(* IEC 61131-3 sources: SRCI/RobotLibrary/RobotLibrary/POUs/SearchHardstop/MC_SearchHardStop, 1 file *)

(* ---- MC_SearchHardStopFB.st ---- *)
/// Move robot into contact with obstruction (mechanical Limit) and hold it in this position
FUNCTION_BLOCK MC_SearchHardStopFB EXTENDS RobotLibraryBaseExecuteFB
// -------------------------------------------------------------------------
//  SRCI Robot Library
// -------------------------------------------------------------------------
//
//  Object:      SearchHardStopFB
//  Author:      Thorsten Brach
//  Date:        2024-06-01
//
//  Description:
//
//
//  Copyright:
//    (C) 2024 Thorsten Brach. All rights reserved
//             Licensed under the LGPL-3.0 license.
//
//  Disclaimer:
//    This project is provided without any guarantee and can be used for
//    private and commercial purposes. Any use is at the user’s
//    own risk and responsibility.
//
// -------------------------------------------------------------------------
VAR_INPUT
  /// Parameter which determines the behavior towards the previously sent and still active or buffered commands
  AbortingMode       : AbortingMode;
  /// Defines the target sequence in which the command will be executed
  SequenceFlag       : SequenceFlag;
  /// command parameter
  ParCmd             : SearchHardStopParCmd;
END_VAR

VAR_OUTPUT
  /// Command is transferred and confirmed by the RC
  CommandBuffered    : BOOL;
  /// The command takes control of the motion of the according axis group
  Active             : BOOL;
  /// The command was aborted by another command.
  CommandAborted     : BOOL;
  /// TRUE, while command is interrupted during execution and can be continued
  CommandInterrupted : BOOL;
  /// command results
  OutCmd             : SearchHardStopOutCmd;
END_VAR

VAR
  /// internal copy of command parameter
 _parCmd             : SearchHardStopParCmd;
  /// command data to send
 _command            : SearchHardStopSendData;
  /// response data received
 _response           : SearchHardStopRecvData;
END_VAR

  SUPER^(AxesGroup := AxesGroup);

END_FUNCTION_BLOCK

METHOD CheckParameterChanged : BOOL
VAR_IN_OUT
  /// Robot assignment of function
  AxesGroup    : AxesGroup;
END_VAR

  // Check ParCmd Size is > 0, becaue MemCmp does not work correctly with size = 0
  IF (SIZEOF(ParCmd) = 0)
  THEN
    RETURN;
  END_IF

  // compare memory
  CheckParameterChanged := ( MemCmp(ADR(ParCmd), ADR(_parCmd), SIZEOF(ParCmd)) <> RobotLibraryConstants.OK );

  IF ( CheckParameterChanged )
  THEN
    // update internal copy of parameters
   _parCmd := ParCmd;
    // inc parameter sequence
   _command.ParSeq := _command.ParSeq + 1;
    // update command data
    CommandData := CreateCommandPayload(); // ( Access via reference to rCommandFB in ACR )
    // notify active command register
    AxesGroup.Acyclic.ActiveCommandRegister.NotifyParameterChanged := _uniqueID;
  END_IF

END_METHOD

METHOD INTERNAL CreateCommandPayload : SendData
// Table 6-405: Sent CMD payload (PLC to RC) of "SearchHardStop"
// --------------------------
// Header
// --------------------------
// Byte 00 : UINT  - Type HB
// Byte 01 :       - Type LB
// Byte 02 : USINT - Reserve | ExecutionMode
// Byte 03 : USINT - ParSeq  | Priority
// --------------------------
// Datablock
// --------------------------
 // Byte 04 : UINT  VelocityRate;
 // Byte 05 :       VelocityRate;
 // Byte 06 : UINT  AccelerationRate;
 // Byte 07 :       AccelerationRate;
 // Byte 08 : UINT  DecelerationRate;
 // Byte 09 :       DecelerationRate;
 // Byte 10 : UINT  JerkRate;
 // Byte 11 :       JerkRate;
 // Byte 12 : USINT ToolNo;
 // Byte 13 : USINT FrameNo;
 // Byte 14 : REAL  Position.X;
 // Byte 15 :       Position.X;
 // Byte 16 :       Position.X;
 // Byte 17 :       Position.X;
 // Byte 18 : REAL  Position.Y;
 // Byte 19 :       Position.Y;
 // Byte 20 :       Position.Y;
 // Byte 21 :       Position.Y;
 // Byte 22 : REAL  Position.Z;
 // Byte 23 :       Position.Z;
 // Byte 24 :       Position.Z;
 // Byte 25 :       Position.Z;
 // Byte 26 : REAL  Position.RX;
 // Byte 27 :       Position.RX;
 // Byte 28 :       Position.RX;
 // Byte 29 :       Position.RX;
 // Byte 30 : REAL  Position.RY;
 // Byte 31 :       Position.RY;
 // Byte 32 :       Position.RY;
 // Byte 33 :       Position.RY;
 // Byte 34 : REAL  Position.RZ;
 // Byte 35 :       Position.RZ;
 // Byte 36 :       Position.RZ;
 // Byte 37 :       Position.RZ;
 // Byte 38 : BYTE  - - - - - W E S;
 // Byte 39 : BYTE  Reserved;
 // Byte 40 : BYTE  Position.TurnNumber[0];
 // Byte 41 : BYTE  Position.TurnNumber[1];
 // Byte 42 : BYTE  Position.TurnNumber[2];
 // Byte 43 : BYTE  Position.TurnNumber[3];
 // Byte 44 : REAL  Position.E1;
 // Byte 45 :       Position.E1;
 // Byte 46 :       Position.E1;
 // Byte 47 :       Position.E1;
 // Byte 48 : USINT OriMode;
 // Byte 49 : USINT DetectionMode;
 // Byte 50 : BOOL  Manipulation;
 // Byte 51 : BYTE  Reserved;
 // Byte 52 : REAL  DetectionVector[0];
 // Byte 53 :       DetectionVector[0];
 // Byte 54 :       DetectionVector[0];
 // Byte 55 :       DetectionVector[0];
 // Byte 56 : REAL  DetectionVector[1];
 // Byte 57 :       DetectionVector[1];
 // Byte 58 :       DetectionVector[1];
 // Byte 59 :       DetectionVector[1];
 // Byte 60 : REAL  DetectionVector[2];
 // Byte 61 :       DetectionVector[2];
 // Byte 62 :       DetectionVector[2];
 // Byte 63 :       DetectionVector[2];
 // Byte 64 : REAL  DetectionVector[3];
 // Byte 65 :       DetectionVector[3];
 // Byte 66 :       DetectionVector[3];
 // Byte 67 :       DetectionVector[3];
 // Byte 68 : REAL  DetectionVector[4];
 // Byte 69 :       DetectionVector[4];
 // Byte 70 :       DetectionVector[4];
 // Byte 71 :       DetectionVector[4];
 // Byte 72 : REAL  DetectionVector[5];
 // Byte 73 :       DetectionVector[5];
 // Byte 74 :       DetectionVector[5];
 // Byte 75 :       DetectionVector[5];
 // Byte 76 : BYTE  ConfigMode[0];
 // Byte 77 : BYTE  ConfigMode[1];
 // Byte 78 : USINT TurnMode;
 // Byte 79 : REAL  Position.E2;
 // Byte 80 :       Position.E2;
 // Byte 81 :       Position.E2;
 // Byte 82 :       Position.E2;
 // Byte 83 : REAL  Position.E3;
 // Byte 84 :       Position.E3;
 // Byte 85 :       Position.E3;
 // Byte 86 :       Position.E3;
 // Byte 87 : REAL  Position.E4;
 // Byte 88 :       Position.E4;
 // Byte 89 :       Position.E4;
 // Byte 90 :       Position.E4;
 // Byte 91 : REAL  Position.E5;
 // Byte 92 :       Position.E5;
 // Byte 93 :       Position.E5;
 // Byte 94 :       Position.E5;
 // Byte 95 : REAL  Position.E6;
 // Byte 96 :       Position.E6;
 // Byte 97 :       Position.E6;
 // Byte 98 :       Position.E6;

  // set command parameter
  _command.CmdTyp           :=  CmdType.SearchHardstop;
  _command.ExecMode         :=  ExecMode;
  _command.ParSeq           := _command.ParSeq;
  _command.Priority         :=  Priority;
  _command.VelocityRate     := REAL_TO_UINT(_parCmd.VelocityRate     * RobotLibraryConstants.REAL_CONVERSION_FACTOR);
  _command.AccelerationRate := REAL_TO_UINT(_parCmd.AccelerationRate * RobotLibraryConstants.REAL_CONVERSION_FACTOR);
  _command.DecelerationRate := REAL_TO_UINT(_parCmd.DecelerationRate * RobotLibraryConstants.REAL_CONVERSION_FACTOR);
  _command.JerkRate         := REAL_TO_UINT(_parCmd.JerkRate         * RobotLibraryConstants.REAL_CONVERSION_FACTOR);
  _command.ToolNo           := _parCmd.ToolNo;
  _command.FrameNo          := _parCmd.FrameNo;
  _command.Position         := _parCmd.Position;
  _command.OriMode          := _parCmd.OriMode;
  _command.DetectionMode    := _parCmd.DetectionMode;
  _command.Manipulation     := _parCmd.Manipulation;
  _command.Reserve          :=  0;
  _command.DetectionVector  := _parCmd.DetectionVector;
  _command.ConfigMode[0].0   := _parCmd.ConfigMode.Shoulder.0;
  _command.ConfigMode[0].1   := _parCmd.ConfigMode.Shoulder.1;
  _command.ConfigMode[0].2   := _parCmd.ConfigMode.Shoulder.2;
  _command.ConfigMode[0].3   := _parCmd.ConfigMode.Shoulder.3;
  _command.ConfigMode[0].4   := _parCmd.ConfigMode.Elbow.0;
  _command.ConfigMode[0].5   := _parCmd.ConfigMode.Elbow.1;
  _command.ConfigMode[0].6   := _parCmd.ConfigMode.Elbow.2;
  _command.ConfigMode[0].7   := _parCmd.ConfigMode.Elbow.3;
  _command.ConfigMode[1].0   := _parCmd.ConfigMode.Wrist.0;
  _command.ConfigMode[1].1   := _parCmd.ConfigMode.Wrist.1;
  _command.ConfigMode[1].2   := _parCmd.ConfigMode.Wrist.2;
  _command.ConfigMode[1].3   := _parCmd.ConfigMode.Wrist.3;
  _command.ConfigMode[1].4   := FALSE;
  _command.ConfigMode[1].5   := FALSE;
  _command.ConfigMode[1].6   := FALSE;
  _command.ConfigMode[1].7   := FALSE;
  _command.TurnMode         := _parCmd.TurnMode;

  // copy command data to header
  _cmdHeader := _command;
  // call base implementation to copy header to payload buffer
  CreateCommandPayload := SUPER^.CreateCommandPayload();

  // add command.VelocityRate
  CreateCommandPayload.AddUint(_command.VelocityRate);
  // add command.AccelerationRate
  CreateCommandPayload.AddUint(_command.AccelerationRate);
  // add command.DecelerationRate
  CreateCommandPayload.AddUint(_command.DecelerationRate);
  // add command.JerkRate
  CreateCommandPayload.AddUint(_command.JerkRate);
  // add command.ToolNo
  CreateCommandPayload.AddUsint(_command.ToolNo);
  // add command.FrameNo
  CreateCommandPayload.AddUsint(_command.FrameNo);
  // add command.Position.X
  CreateCommandPayload.AddReal(_command.Position.X);
  // add command.Position.Y
  CreateCommandPayload.AddReal(_command.Position.Y);
  // add command.Position.Z
  CreateCommandPayload.AddReal(_command.Position.Z);
  // add command.Position.Rx
  CreateCommandPayload.AddReal(_command.Position.Rx);
  // add command.Position.Ry
  CreateCommandPayload.AddReal(_command.Position.Ry);
  // add command.Position.Rz
  CreateCommandPayload.AddReal(_command.Position.Rz);
  // add command.Position.Config
  CreateCommandPayload.AddArmConfig(_command.Position.Config);
  // add command.Position.TurnNumber
  CreateCommandPayload.AddTurnNumber(_command.Position.TurnNumber);
  // add command.Position.E1
  CreateCommandPayload.AddReal(_command.Position.E1);
  // add command.OriMode
  CreateCommandPayload.AddUsint(_command.OriMode);
  // add command.DetectionMode
  CreateCommandPayload.AddUsint(_command.DetectionMode);
  // add command.Manipulation
  CreateCommandPayload.AddBool(_command.Manipulation);
  // add command.Reserve
  CreateCommandPayload.AddByte(_command.Reserve);
  // add command.DetectionVector[0]
  CreateCommandPayload.AddReal(_command.DetectionVector[0]);
  // add command.DetectionVector[1]
  CreateCommandPayload.AddReal(_command.DetectionVector[1]);
  // add command.DetectionVector[2]
  CreateCommandPayload.AddReal(_command.DetectionVector[2]);
  // add command.DetectionVector[3]
  CreateCommandPayload.AddReal(_command.DetectionVector[3]);
  // add command.DetectionVector[4]
  CreateCommandPayload.AddReal(_command.DetectionVector[4]);
  // add command.DetectionVector[5]
  CreateCommandPayload.AddReal(_command.DetectionVector[5]);
  // add command.ConfigMode[0]
  CreateCommandPayload.AddByte(_command.ConfigMode[0]);
  // add command.ConfigMode[1]
  CreateCommandPayload.AddByte(_command.ConfigMode[1]);
  // add command.TurnMode
  CreateCommandPayload.AddUsint(_command.TurnMode);
  // add command.Position.E2
  CreateCommandPayload.AddReal(_command.Position.E2);
  // add command.Position.E3
  CreateCommandPayload.AddReal(_command.Position.E3);
  // add command.Position.E4
  CreateCommandPayload.AddReal(_command.Position.E4);
  // add command.Position.E5
  CreateCommandPayload.AddReal(_command.Position.E5);
  // add command.Position.E6
  CreateCommandPayload.AddReal(_command.Position.E6);

END_METHOD

METHOD FB_init : BOOL
VAR_INPUT
  /// if TRUE, the retain variables are initialized (warm start / cold start)
	bInitRetains : BOOL;
  /// if TRUE, the instance afterwards gets moved into the copy code (online change)
	bInCopyCode  : BOOL;
END_VAR

  MyType := 'MC_SearchHardStopFB';

END_METHOD

METHOD PROTECTED OnCall
VAR_IN_OUT
  /// Robot assignment of function
  AxesGroup : AxesGroup;
END_VAR

  // call base implementation
  SUPER^.OnCall(AxesGroup := AxesGroup);

  CASE _stepCmd OF

    00:  IF ( _execute_R.Q )
         THEN
           // set busy flag
           Busy := TRUE;
           // Reset command outputs
           MemSet(ADR(OutCmd),0,SIZEOF(OutCmd));
           // apply command parameter
          _parCmd := ParCmd;
           // init parameter sequence
          _command.ParSeq := 1;
           // set timeout
           SetTimeout(PT := _timeoutCmd, rTimer := _timerCmd);
           // inc step counter
          _stepCmd := _stepCmd + 1;
  	     END_IF

    01:  // create command data
         CommandData := CreateCommandPayload();
         // Add command to active command register
        _uniqueID := AxesGroup.Acyclic.ActiveCommandRegister.AddCmd( pCommandFB := ADR(THIS^ ));
         // set timeout
         SetTimeout(PT := _timeoutCmd, rTimer := _timerCmd);
         // inc step counter
        _stepCmd := _stepCmd + 1;

    02:  // Wait for responce received
         IF ( _responseReceived )
         THEN
           // reset response received flag
          _responseReceived := FALSE;
           // reset Active flag
           Active := FALSE;

           CASE  _response.State
           OF
             CmdMessageState.BUFFERED    : CommandBuffered    := TRUE;
             CmdMessageState.ACTIVE      : Active             := TRUE;
             CmdMessageState.INTERRUPTED : CommandInterrupted := TRUE;
             CmdMessageState.DONE        : Done               := TRUE;
             CmdMessageState.ABORTED     : CommandAborted     := TRUE;
             CmdMessageState.ERROR       : Error              := TRUE;
  				 END_CASE

           // Done, Aborted or Error ?
           IF (_response.State >= CmdMessageState.DONE )
           THEN
             // Reset Busy flag
             Busy := FALSE;
             // Update results
             OutCmd.InClamping        := _response.InClamping;
             OutCmd.Progress          := _response.Progress;
             OutCmd.RemainingDistance := _response.RemainingDistance;
             // set timeout
             SetTimeout(PT := _timeoutCmd, rTimer := _timerCmd);
             // inc step counter
            _stepCmd := _stepCmd + 1;
  				 END_IF
         END_IF

    03: IF ( NOT Execute)
        THEN
          Reset();
  			END_IF
  ELSE
    // invalid step
    ErrorID := RobotLibraryEvents.ERR_INVALID_STEP;
  END_CASE

  // Cancel
  IF (Busy) AND (NOT Execute)
  THEN
    // try to remove cmd
    AxesGroup.Acyclic.ActiveCommandRegister.RemoveCmd(_uniqueID);
  END_IF

  // Reset FB
  IF ( NOT Execute )
  THEN
    Reset();
  END_IF

END_METHOD

METHOD INTERNAL ParseResponsePayload : DINT
// Table 6-406: Received CMD payload (RC to PLC) of "SearchHardStop"
// --------------------------
// Header
// --------------------------
// Byte 00 : USINT   - ParSeq | State
// Byte 01 : SINT    - AlarmMessageSeverity
// Byte 02 : UINT    - AlarmMessageCode HB
// Byte 03 :         - AlarmMessageCode LB
// --------------------------
// Datablock
// --------------------------
// Byte 04 : UINT    - Progress LW HB
// Byte 05 :         - Progress LW LB
// Byte 06 : REAL    - RemainingDistance HW HB
// Byte 07 :         - RemainingDistance HW LB
// Byte 08 :         - RemainingDistance LW HB
// Byte 09 :         - RemainingDistance LW LB
// Byte 10 : BOOL    - InClamping
VAR_INPUT
  /// Response data
  ResponseData : RecvData;
END_VAR

  // call base implementation to parse the header from payload buffer
  ResponseData.PayloadPtr := SUPER^.ParseResponsePayload(ResponseData);

  // copy parsed header to response
  _response.ParSeq               := _rspHeader.ParSeq;
  _response.State                := _rspHeader.State;
  _response.AlarmMessageSeverity := _rspHeader.AlarmMessageSeverity;
  _response.AlarmMessageCode     := _rspHeader.AlarmMessageCode;

  // Get Response.Progress
  _response.Progress := ResponseData.GetUint();
  // Get Response.RemainingDistance
  _response.RemainingDistance := ResponseData.GetReal();
  // Get Response.InClamping
  _response.InClamping := ResponseData.GetBool();

END_METHOD

METHOD PROTECTED Reset : DINT
VAR_INPUT
END_VAR

  Reset := SUPER^.Reset();

  Done               := FALSE;
  Busy               := FALSE;
  Active             := FALSE;
  CommandBuffered    := FALSE;
  CommandAborted     := FALSE;
  CommandInterrupted := FALSE;

END_METHOD
